Universal Robots PolyScope program: roof_a.urp

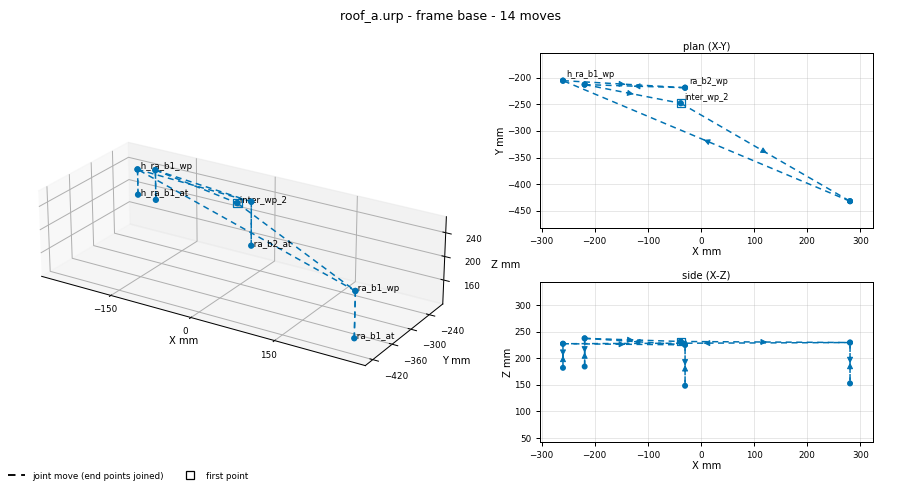
[picture p0: tool path of roof_a.urp in frame base, 14 of 14 moves have a stored position in this frame; points joined in program order, loops and branches not executed]
Program roof_a (installation=default directory=/programs/Session 1 createdIn=5.3.1.64192 lastSavedIn=5.3.1.64192 robotSerialNumber=20195300365)
Calibrated DH parameters: a=[-0.000093, -0.190649, -0.212673, 0.000091, -0.000205, 0]; d=[0.151591, 44.061648, -42.488068, -1.442789, 0.085322, 0.091911]; alpha=[1.570082, -0.003447, 0.007513, 1.572293, -1.571904, 0]; deltaTheta=[0, -0.672656, 0.728185, -0.055522, 0.000005, 0]
Robot Program (runOnlyOnce=true)
  URCap Gripper Activate (Robotiq_Grippers, Robotiq Inc.) dataModel(ResetAndActivateKey=false)
  URCap Gripper (Robotiq_Grippers, Robotiq Inc.) dataModel(position=50.0, force=100.0, speed=100.0, positionInDouble=50.0, forceInDouble=100.0, speedInDouble=100.0, slaveIds=[9], blocking=true)
  MoveJ speed 60 deg/s, acceleration 80 deg/s^2 (useActiveTCP=true) feature=Base
    Waypoint inter_wp_2: TCP in base x=-38.107 y=-247.898 z=231.572 mm, rx=2.241 ry=2.1798 rz=0.019 rad; joints [-68.076, -72.135, -124.793, -72.457, 91.361, -246.109] deg
  Folder Roof_A
    MoveJ speed 60 deg/s, acceleration 80 deg/s^2 (useActiveTCP=true) feature=Base
      Waypoint ra_b1_wp: TCP in base x=280.355 y=-432.175 z=229.592 mm, rx=2.2498 ry=2.1383 rz=0.0086 rad; joints [-42.341, -144.4, -29.155, -94.202, 90.433, -219.411] deg
      Waypoint ra_b1_at: TCP in base x=280.345 y=-432.185 z=152.652 mm, rx=2.2498 ry=2.1383 rz=0.0087 rad; joints [-42.387, -145.97, -46.929, -74.856, 90.432, -219.319] deg
      URCap Gripper (Robotiq_Grippers, Robotiq Inc.) dataModel(position=100.0, force=100.0, speed=100.0, positionInDouble=100.0, forceInDouble=100.0, speedInDouble=100.0, slaveIds=[9], blocking=true)
      Waypoint ra_b1_wp: TCP in base x=280.355 y=-432.175 z=229.592 mm, rx=2.2498 ry=2.1383 rz=0.0086 rad; joints [-42.341, -144.4, -29.155, -94.202, 90.433, -219.411] deg
      Waypoint h_ra_b1_wp: TCP in base x=-259.638 y=-205.368 z=227.372 mm, rx=2.9429 ry=-0.031 rz=-0.0033 rad; joints [-120.289, -93.82, -112.087, -54.007, 95.739, -208.146] deg
      Waypoint h_ra_b1_at: TCP in base x=-259.633 y=-205.356 z=182.009 mm, rx=2.9429 ry=-0.031 rz=-0.0033 rad; joints [-120.304, -100.149, -119.184, -40.582, 95.664, -208.103] deg
      URCap Gripper (Robotiq_Grippers, Robotiq Inc.) dataModel(position=50.0, force=100.0, speed=100.0, positionInDouble=50.0, forceInDouble=100.0, speedInDouble=100.0, slaveIds=[9], blocking=true)
      Waypoint h_ra_b1_wp: TCP in base x=-259.638 y=-205.368 z=227.372 mm, rx=2.9429 ry=-0.031 rz=-0.0033 rad; joints [-120.289, -93.82, -112.087, -54.007, 95.739, -208.146] deg
    MoveJ speed 60 deg/s, acceleration 80 deg/s^2 (useActiveTCP=true) feature=Base
      Waypoint ra_b2_wp: TCP in base x=-29.938 y=-218.629 z=225.3 mm, rx=-2.2436 ry=-2.1936 rz=-0.0198 rad; joints [-62.186, -62.499, -131.394, -76.453, 91.059, -240.54] deg
      Waypoint ra_b2_at: TCP in base x=-29.954 y=-218.613 z=148.235 mm, rx=-2.2436 ry=-2.1934 rz=-0.0198 rad; joints [-62.247, -75.96, -148.106, -46.285, 90.919, -240.408] deg
      URCap Gripper (Robotiq_Grippers, Robotiq Inc.) dataModel(position=100.0, force=100.0, speed=100.0, positionInDouble=100.0, forceInDouble=100.0, speedInDouble=100.0, slaveIds=[9], blocking=true)
      Waypoint ra_b2_wp: TCP in base x=-29.938 y=-218.629 z=225.3 mm, rx=-2.2436 ry=-2.1936 rz=-0.0198 rad; joints [-62.186, -62.499, -131.394, -76.453, 91.059, -240.54] deg
      Waypoint h_ra_b2_wp: TCP in base x=-218.822 y=-212.79 z=237.473 mm, rx=0.0119 ry=3.1066 rz=-0.2822 rad; joints [-112.389, -86.229, -116.282, -58.23, 95.353, -381.095] deg
      Waypoint h_ra_b2_at: TCP in base x=-218.835 y=-212.79 z=184.432 mm, rx=0.012 ry=3.1067 rz=-0.2822 rad; joints [-112.412, -93.62, -125.525, -41.59, 95.263, -381.034] deg
      URCap Gripper (Robotiq_Grippers, Robotiq Inc.) dataModel(position=50.0, force=100.0, speed=100.0, positionInDouble=50.0, forceInDouble=100.0, speedInDouble=100.0, slaveIds=[9], blocking=true)
      Waypoint h_ra_b2_wp: TCP in base x=-218.822 y=-212.79 z=237.473 mm, rx=0.0119 ry=3.1066 rz=-0.2822 rad; joints [-112.389, -86.229, -116.282, -58.23, 95.353, -381.095] deg
  MoveJ speed 60 deg/s, acceleration 80 deg/s^2 (useActiveTCP=true) feature=Base
    Waypoint inter_wp_2: TCP in base x=-38.107 y=-247.898 z=231.572 mm, rx=2.241 ry=2.1798 rz=0.019 rad; joints [-68.076, -72.135, -124.793, -72.457, 91.361, -246.109] deg
